Staubli VAL3: getSize.pgx

public program getSize(num& x_nSize[])
  local string l_sType
begin
  //
end
